Staubli VAL3: Main_app.dtx

bool bBooltoNum
bool bBtnCtrlOpc
bool bBtnIntercambio
bool bError
public bool bEstAtornillador = true
public bool bEstPinza = true
public bool bHerramientaRobot = true
bool bOk
public bool bTLocked
public bool bTUnlocked = true
public bool btnToolChangeBolt
public bool btnToolChangeGrip
bool validPos
dio dChangerValve = {link=ValveIO\valve1}
dio dDioEstAtornillador = {link=CE061C2D-63EF-47EF-A59E-9D0AF6F8F85C}
dio dDioEstPinza = {link=09F12A79-E04E-419B-9AAF-7725DDDBD1AC}
dio dDioHerramientaRobot = {link=7E390559-96A8-403A-B445-689BBF355DEA}
dio dDioTLocked = {link=F2CD6568-BB9E-49C8-A7B4-91D8A66F9C51}
dio dDioTUnlocked = {link=60862B78-E473-4D73-B0A1-35126C8FEF27}
frame fHaption = {x=107.807516, y=-386.531428, z=887.560715, rx=-89.0477411, ry=-149.698587, rz=0.421407, fatherId=world[0]}
frame fToolChange = {x=615.030242, y=458.213417, z=150.671162, rx=-90.0936151, ry=30.458364, rz=89.118179, fatherId=world[0]}
jointRx jChange = {j1=-4.0714236, j2=-3.552111, j3=129.273225, j4=106.087665, j5=68.799532, j6=6.346847}
jointRx jHome = {j1=57.800006, j2=-37.780028, j3=119.215944, j4=179.0580443, j5=81.384924, j6=-131.0356711}
public jointRx jInitial = {j1=57.800006, j2=-37.780028, j3=119.215944, j4=179.0580443, j5=81.384924, j6=-131.0356711}
public jointRx jJointRx
jointRx jResult
jointRx jTouch = {j1=60.497505, j2=-107.87914, j3=120.00337332, j4=178.372552, j5=-48.125989, j6=4.636406}
mdesc mAppro = {accel=5, vel=5, decel=5, leave=1, reach=1}
mdesc mChange = {accel=10, vel=10, decel=10, leave=10, reach=10}
mdesc mNomSpeed = {accel=50, vel=50, decel=50}
public num OPCf1
public num OPCf2
public num OPCf3
public num OPCf4
public num OPCf5
public num OPCf6
public num OPCj1
public num OPCj2
public num OPCj3
public num OPCj4
public num OPCj5
public num OPCj6
public num OPCrx
public num OPCry
public num OPCrz
public num OPCx
public num OPCy
public num OPCz
num nCmd[6]
num nCmdTrans[6]
num nI
num nJ
public num nListForces[6]
num nPos
num nRawUdp[48]
num nState
num nTemp
public pointRx pActualPos
pointRx pPointRx
pointRx pTest = {x=-252.530153, y=263.294912, z=427.370916, rx=5.121571, ry=-7.129797, rz=162.640171}
pointRx pTool1 = {x=26.46, y=-161.846445, z=25.66398, rx=0.739769, ry=-0.0144029, rz=-134.866663, shoulder=lefty, elbow=epositive, wrist=wpositive, fatherId=fToolChange[0]}
pointRx pTool2 = {x=24.417771, y=213.35041, z=25.529958, rx=-0.30514, ry=-0.197907, rz=46.419643, shoulder=lefty, elbow=epositive, wrist=wpositive, fatherId=fToolChange[0]}
string sInfo = "Cogiendo el atornillador."
string sOutput = "No se ha podido dar potencia al brazo"
string sStringRaw[48]
tool tAtornillador = {x=-0.0903, y=-165.0894, z=43.1596, fatherId=tChanger[0]}
tool tChanger = {z=62.5, fatherId=flange[0], ioLink=ValveIO\valve1, ioOpen=0.5, ioClose=0.5}
tool tPinza = {y=48.1055, z=146.1642, fatherId=tChanger[0]}
tool tPuntero = {z=118, fatherId=flange[0]}
tool tTeach = {z=90, fatherId=flange[0]}
jointRx jGimbal = {j6=1}
public num nSpeedRate
public dio dDioMoveGripper = {link=B2194EAF-1145-4C79-9BA9-5960C08FF7FC}
public bool bMoveGripper
public bool bLockRotation
public bool bManualJoint
public bool bModeChanged
public num OPCj1cmd
public num OPCj2cmd
public num OPCj3cmd
public num OPCj4cmd
public num OPCj5cmd
public num OPCj6cmd
public bool bCogerPinza
public bool bCogerAtornillador
public bool bDejarPinza
public bool bDejarAtornillador
jointRx jStart = {j1=-6.36110936292703E-15, j2=4.98, j3=-90.18, j4=1.4230002260189E-21, j5=85.08, j6=6.36110860462371E-15}
bool bSupervisor
num countstring
num countrecord
bool flagactive
num lastReceived
dio dDioDoor1Status = {link=7E2C1981-2091-4168-A4C7-3B8F54F93892}
dio dDioDoor2Status = {link=DD4B0AAB-BB16-4B26-8EC1-F4B17697477E}
dio dDioEmergencyButton = {link=70CCD0F6-6BE7-4533-984C-B059D9950979}
dio dESbutton = {link=Rsi9IO\IusoA1}
dio dDoor1 = {link=Rsi9IO\IusiB1}
dio dDoor2 = {link=Rsi9IO\IusiA1}
num nStart
num nDelay
public dio diJ207J208_RE_PNS_I6 = {link=09F12A79-E04E-419B-9AAF-7725DDDBD1AC}
public dio doJ207J208_RE_PNS_Q6 = {link=5F8C0500-A0C2-418B-B33F-DA7D83872BF3}
public dio diJ207J208_RE_PNS_I2 = {link=60862B78-E473-4D73-B0A1-35126C8FEF27}
public dio doJ207J208_RE_PNS_Q5 = {link=70CCD0F6-6BE7-4533-984C-B059D9950979}
public dio doJ207J208_RE_PNS_Q3 = {link=7E2C1981-2091-4168-A4C7-3B8F54F93892}
public dio diJ207J208_RE_PNS_I1 = {link=7E390559-96A8-403A-B445-689BBF355DEA}
public dio diJ207J208_RE_PNS_I5 = {link=826855D7-B3BE-4D72-B5FB-E89AA8CE1BC8}
public dio doJ207J208_RE_PNS_Q7 = {link=89E313F4-BC69-4F53-99A0-AECEC5F380AE}
public dio doJ207J208_RE_PNS_Q2 = {link=8EED7CAF-566F-42FA-AB95-4CE736BA248A}
public dio doJ207J208_RE_PNS_Q1 = {link=957CEE52-2BF5-4DF0-8E67-FA620ACF6C14}
public dio doJ207J208_RE_PNS_Q0 = {link=B2194EAF-1145-4C79-9BA9-5960C08FF7FC}
public dio diJ207J208_RE_PNS_I7 = {link=CE061C2D-63EF-47EF-A59E-9D0AF6F8F85C}
public dio diJ207J208_RE_PNS_I4 = {link=D971BF12-E116-4771-AC73-77C32A945796}
public dio doJ207J208_RE_PNS_Q4 = {link=DD4B0AAB-BB16-4B26-8EC1-F4B17697477E}
public dio diJ207J208_RE_PNS_I3 = {link=ECDEAE6F-FADA-4468-909E-1E4B6F2B874F}
public dio diJ207J208_RE_PNS_I0 = {link=F2CD6568-BB9E-49C8-A7B4-91D8A66F9C51}
public sio SocketTCP = {link=Socket\ReceiveTcp}
public sio SocketUDP = {link=UdpSocket\ReceiveUdp}
num desordenados
num OpcPrecisionMovement
trsf trAlter
num nAlterBeginState
pointRx pFinishAlter = {x=-336.628720241718, y=50, z=505.159108540589, rx=-5.05493480877665E-23, ry=1.40872651758736E-05, rz=-1.15631870617668E-21, shoulder=righty, elbow=enegative, wrist=wpositive, fatherId=world[0]}
trsf trAlterMove
num OpcStepsMovement
num nAlterState
num nAlterEndState
pointRx pStart = {x=-336.829738845272, y=49.9999961803571, z=558.957317821961, rx=2.83367334814845E-09, ry=-0.115117715818688, rz=2.8115150816022E-12, shoulder=righty, elbow=enegative, wrist=wpositive, fatherId=world[0]}
num nRecordCmd[2010 3]
num nRecordCmdX[10000]
num nRecordCmdY[10000]
num nRecordCmdID[10000]
string sStringHistorical[10000]
bool almacenar
sio SocketUDPForceSensor = {link=UdpSocket\SocketUDPForceSensor}
num nRequestUDP[8]
num nrxforce
num nDiagSocket
num nDiagSocket2
num nResponseUDP[36]
num nResponses
num Fx
num Fy
num Fz
num Tx
num Ty
num Tz
num nTestfB[36]
num nTestfBIN[288]
num i
num bytenum
num cociente
num resto
num HEXNUMBER[4 2]
num DECNUMBER
num j
num FxLimit
num FyLimit
num FzLimit
num TxLimit
num TyLimit
num TzLimit
bool followHuman
bool bSupervisorForce
pointRx pPress1 = {x=-336.870168433842, y=49.999992370606, z=579.007588648422, rx=2.8335220482869E-09, ry=-0.115113873837275, rz=2.84048267905755E-12, shoulder=righty, elbow=enegative, wrist=wpositive, fatherId=world[0]}
pointRx pRelease1 = {x=-336.829643365744, y=-50.1476616059199, z=558.909800775024, rx=-9.93639403181191E-07, ry=-0.115115185933709, rz=-9.61953709022073E-07, shoulder=righty, elbow=enegative, wrist=wpositive, fatherId=world[0]}
pointRx pPress2 = {x=-336.870134367357, y=-50.1476774705417, z=578.993918901558, rx=-2.56189918387667E-06, ry=-0.115109572206669, rz=-2.47515326511544E-06, shoulder=righty, elbow=enegative, wrist=wpositive, fatherId=world[0]}
pointRx pRelease2 = {x=-336.829650546973, y=-150.228261555763, z=558.909800434958, rx=-1.72565131768918E-06, ry=-0.11511397198566, rz=-1.69662426766672E-06, shoulder=righty, elbow=enegative, wrist=wpositive, fatherId=world[0]}
pointRx pPress3 = {x=-336.86978960782, y=-150.228255444793, z=578.871206987795, rx=-3.03400370196542E-07, ry=-0.115116778365496, rz=-2.63029287251087E-06, shoulder=righty, elbow=enegative, wrist=wpositive, fatherId=world[0]}
string sOPCRobotyReady
bool OpcPreciseMode
pointRx pSlide1 = {x=197.7, y=-267.76, z=591.67, rz=17.74, fatherId=world[0]}
pointRx pSlide2 = {x=-197.7, y=-267.76, z=595.22, rz=17.74, fatherId=world[0]}
pointRx pSlide3 = {x=-269.92, y=-408.17, z=595.21, rz=17.74, fatherId=world[0]}
sio SocketUDPMySensor = {link=UdpSocket\SocketUDPMySensor}
public num FxFlag
public num FyFlag
public num FzFlag
num OPCrxcmdOut
num OPCrycmdOut
num OPCrzcmdOut
num OpcStepsRotation
bool OPCGoHoming
bool OpcPreciseModePrevious
num auxencod
num nReplyMySensor[24]
public bool OPCChangeTool
bool flagOnceChangeTool
bool flagAlter
bool launchAlter
bool launchManualJoint
bool launchToolChange
jointRx jHere
bool OPCSetZeroForces
bool prevlaunchAlter
bool prevlaunchManualJoint
bool prevlaunchToolChange
jointRx jResumeAlter = {j2=4.98, j3=-90.18, j5=85.08}
